Staubli VAL3: getItem_num.pgx

public program getItem_num(string& x_sItem (dimensions=1), string x_sId (dimensions=1))
begin
  // get the name
  if isDefined(cCount[x_sId])
    x_sItem=cCount[x_sId].sName
  elseIf isDefined(aCount[x_sId])
    x_sItem=aCount[x_sId].sName
  endIf
end
